(* CODESYS project PS_DcUpsEC_3.library
   Author: SAC
   Placeholder: PS_DcUpsEC
   Title: PS_DcUpsEC
   Version: 3.0
   Description: Function blocks for DC Uninterruptible Power Supplies with EtherCAT Interface
   Company: Phoenix Contact GmbH & Co.KG

Project tree, tasks and I/O mapping:
  libraries: Tc2_EtherCAT, * (Beckhoff Automation GmbH); Tc2_Standard, * (Beckhoff Automation GmbH); Tc2_System, * (Beckhoff Automation GmbH); Tc3_Module, * (Beckhoff Automation GmbH)
  DUTs/
    data type PS_CYCLIC_DATA
    data type PS_STATUS_FUNCTIONS
    data type PS_STATUS_INTERFACE
  GVLs/
  POUs/
    function block PS_Q4_DcUpsEC_Cyclic_3 [ST]: NewAlarmHandling, OldAlarmHandling
    function block PS_Q4_DcUpsEC_Param_1 [ST]
  Version/
    global variables Global_Version
  VISUs/
*)

// DUTs/PS_CYCLIC_DATA
TYPE PS_CYCLIC_DATA :
STRUCT
	srStatus_Functions  : PS_STATUS_FUNCTIONS;  (*Collection OF status signals*)        
	srStatus_Interface  : PS_STATUS_INTERFACE;  (*Collection OF interface signals*)        
	wInputVoltage       : WORD;         (*Input voltage in mV*)        
	wInputCurrent       : WORD;         (*Input current in mA*)        
	wOutputVoltage      : WORD;         (*Output voltage in mV*)        
	wOutputCurrent      : WORD;         (*Output current in mA*)        
	wBatteryVoltage     : WORD;         (*Battery voltage in mV*)        
	wBatteryChargeCurrent   : WORD;     (*Battery charge current in mA*)        
	wBatteryTemperature     : WORD;     (*Battery temperature in K*)        
	wDeviceTemperature      : WORD;     (*Device temperature in K*)        
	dwSocRemainingTime      : DWORD;    (*Remaining time in seconds*)        
	wSocRemainingTimePC_Shutdown: WORD; (*Remaining time until PC shutdown in s*)        
	wBatRemainingLifetime   : WORD;     (*Remaining lifetime in days*)
END_STRUCT
END_TYPE

// DUTs/PS_STATUS_FUNCTIONS
TYPE PS_STATUS_FUNCTIONS :
STRUCT
	xStartUpActive      : BOOL; (*Device is starting*)        
	xMainPowerModeActive: BOOL; (*Device is in mains mode*)        
	xBatteryModeActive  : BOOL; (*Device is in battery mode*)        
	xOutput             : BOOL; (*Output OF device is on/off*)        
	xBoost              : BOOL; (*Device is in boost mode*)        
	xChargerOn          : BOOL; (*Charger OF device is on/off*)        
	xBatteryComActive   : BOOL; (*Communcation to batteries is active/inactive*)        
	xStatusBatCom       : BOOL; (*Status communcation to batteries: 0=adressing, 1=normal communication*)        
	xAutonomicStart     : BOOL; (*Autonomic start input is open/closed*)        
	xRemoteConnected    : BOOL; (*Remote DI connected/disconnected*)        
	xRemoteEnabled      : BOOL; (*Remote is enabled/disabled*)        
	xPSinBoostMode      : BOOL; (*Power supply is in boost mode*)        
	xPhoenixAddCharger  : BOOL; (*Phoenix Contact additional charger is connected*)        
	xServiceModeActive  : BOOL; (*Device is in service mode*)        
	xBatDelay1Active    : BOOL; (*Battery mode delay time 1 is active*)        
	xBatDelay2Active    : BOOL; (*Battery mode delay time 2 is active*)        
	xBatDelay3Active    : BOOL; (*Battery mode delay time 3 is active**)        
	xExternalCharger    : BOOL; (*External charger active/inactive*)        
	xBufferReady        : BOOL; (*Connected energy storage is ready to buffer*)        
	xButtonUse          : BOOL; (*Service button enabled/disabled*)        
	xSelectorSwitchUse  : BOOL; (*Selector switch enabled/disabled*)        
	xSystemTest         : BOOL; (*System test active/inactive*)        
	xBatCapTest         : BOOL; (*Battery capacity test active/inactive*)        
	xBatteryPresent     : BOOL; (*Energy storage connected/disconnected*)        
	xSOC_Initialized    : BOOL; (*State OF charge initialized*)        
	xTriggerLogData     : BOOL; (*New log data available*)
END_STRUCT
END_TYPE

// DUTs/PS_STATUS_INTERFACE
TYPE PS_STATUS_INTERFACE :
STRUCT
	xDO1            : BOOL; (*DO1 is active/inactive*)        
	xDO2            : BOOL; (*DO2 is active/inactive*)        
	xDO3            : BOOL; (*DO3 is active/inactive*)        
	xDI1            : BOOL; (*DI1 is active/inactive*)        
	xDI2            : BOOL; (*DI2 is active/inactive*)        
	xDI3            : BOOL; (*DI3 is active/inactive*)        
	xModeSelector1  : BOOL; (*mode selector switch 1*)        
	xModeSelector2  : BOOL; (*mode selector switch 2*)        
	xModeSelector3  : BOOL; (*mode selector switch 3*)        
	xModeSelector4  : BOOL; (*mode selector switch 4*)        
	xSwitchPressed  : BOOL; (*Service button pressed/NOT pressed*)        
	xGreenLED       : BOOL; (*Green LED is on/off*)        
	xYellowLED      : BOOL; (*Yellow LED is on/off*)        
	xRedLED         : BOOL; (*Red LED is on/off*)        
	xBargraphRed    : BOOL; (*Red bargraph LED is on/off*)        
	xBargraphGreen1 : BOOL; (*Green bargraph LED 1 is on/off*)        
	xBargraphGreen2 : BOOL; (*Green bargraph LED 2 is on/off*)        
	xBargraphGreen3 : BOOL; (*Green bargraph LED 3 is on/off*)        
	xBargraphGreen4 : BOOL; (*Green bargraph LED 4 is on/off*)        
	xBargraphGreen5 : BOOL; (*Green bargraph LED 5 is on/off*)
	xSFB_Input		: BOOL;	(*SFB input is active/inactive*)
END_STRUCT
END_TYPE

// Version/Global_Version
{attribute 'TcGenerated'}
{attribute 'no-analysis'}
{attribute 'linkalways'}
// This function has been automatically generated from the project information.
VAR_GLOBAL CONSTANT
	{attribute 'const_non_replaced'}
	stLibVersion_PS_DcUpsEC : ST_LibVersion := (iMajor := 3, iMinor := 0, iBuild := 0, iRevision := 0, sVersion := '3.0');
END_VAR

// POUs/PS_Q4_DcUpsEC_Cyclic_3
{attribute 'hide_all_locals'}
FUNCTION_BLOCK PS_Q4_DcUpsEC_Cyclic_3
(*
wDiagCode	wAddDiagCode 	Description
16#0000		16#0000			Function block is inactive
16#8000		16#0000			Function block is active and without errors
*)
VAR_INPUT
	xActivate	: BOOL;		// TRUE: Activates function block
	arrInputPD	: ARRAY [0..30] OF WORD;	// Connect Multilink of TxPDO here
	tTimeout	: TIME := t#15s;	// Timeout value for communication timeout. Default t#15s.
END_VAR
VAR_OUTPUT
	xActive		: BOOL; // TRUE: Function block is working
	xError		: BOOL; // TRUE: An error occured at function block
	wDiagCode	: WORD; // Diagnosis Code of funtcion block error
	wAddDiagCode: WORD;	// Additional information about Diagnosis Code
	wOutputVoltage	: WORD; // Output Voltage of UPS in mV
	wOutputCurrent	: WORD; // Output Current of UPS in mA
	xBatModeActive	: BOOL; // TRUE: UPS is in Battery Mode
	udtDataStruct	: PS_CYCLIC_DATA; // Data structure contains voltages, currents, temperatures and remaining times
	xAlarm : BOOL; // TRUE: An alarm occured on the system
	xWarning : BOOL; // TRUE: An warning occured on the system
	xReplaceBattery : BOOL; // TRUE: Battery has to be replaced
	udtDiag : ARRAY[0..15] OF STRING; // Array of Alarm/Warning messages
END_VAR
VAR 
	(*_xyz - internal variables*)
	_wProcessAlarms : WORD;
	_dwUPSDiagnosis : DWORD;
	_dwBatAlarms : ARRAY[1..5] OF DWORD;
	_dwChargerAlarms : DWORD;
	_nI, _nK, _nM : INT;
	_xWarning: BOOL;
	_xAlarm: BOOL;
	_udtDiag : ARRAY[0..15] OF STRING;;
	_udtDeleteDiag : ARRAY[0..15] OF STRING; 
	_udtDelDataStruct	: PS_CYCLIC_DATA;
	_xBatModeActive: BOOL;
	_xReplaceBattery: BOOL;
	_fbTON : TON;
	_wBatteryVoltageOld	: WORD;
	_wInputVoltageOld : WORD;
	_wInputCurrentOld : WORD;
	_wOutputVoltageOld : WORD;
	_wOutputCurrentOld : WORD;
	_dwSocRemainingTimeOld :DWORD;	
	_xError : BOOL;
	_wDiagCode : WORD;
	_wAddDiagCode : WORD;
	_iNoOfActiveAlarms: INT;
	_iAlarmTypes: INT;
	_iAlarm_ID: INT;
	_iDevice_ID: INT;
	_arrAlarmBuffer : ARRAY [0..15] OF DWORD;
	_xNewAlarm : BOOL;
END_VAR

IF  xActivate THEN
	xActive := TRUE;
	_xError := FALSE;
	_wDiagCode := 16#8000;
	_wAddDiagCode := 16#0000;
	

	//-------------------------------------------------------------------------------
	
	// copy process alarms
	_wProcessAlarms := arrInputPD[16];
	// copy diagnosis alarms
	_dwUPSDiagnosis := SHL(WORD_TO_DWORD(arrInputPD[18]),DWORD#16);;
	_dwUPSDiagnosis := _dwUPSDiagnosis OR WORD_TO_DWORD(arrInputPD[17]);
	// Battery 1 Alarms
	_dwBatAlarms[1] := SHL(WORD_TO_DWORD(arrInputPD[20]),DWORD#16);;
	_dwBatAlarms[1] := _dwBatAlarms[1] OR WORD_TO_DWORD(arrInputPD[19]);
	// Battery 2 Alarms
	_dwBatAlarms[2] := SHL(WORD_TO_DWORD(arrInputPD[22]),DWORD#16);;
	_dwBatAlarms[2] := _dwBatAlarms[2] OR WORD_TO_DWORD(arrInputPD[21]);
	// Battery 3 Alarms
	_dwBatAlarms[3] := SHL(WORD_TO_DWORD(arrInputPD[24]),DWORD#16);;
	_dwBatAlarms[3] := _dwBatAlarms[3] OR WORD_TO_DWORD(arrInputPD[23]);
	// Battery 4 Alarms
	_dwBatAlarms[4] := SHL(WORD_TO_DWORD(arrInputPD[26]),DWORD#16);;
	_dwBatAlarms[4] := _dwBatAlarms[4] OR WORD_TO_DWORD(arrInputPD[25]);
	// Battery 5 Alarms
	_dwBatAlarms[5] := SHL(WORD_TO_DWORD(arrInputPD[28]),DWORD#16);;
	_dwBatAlarms[5] := _dwBatAlarms[5] OR WORD_TO_DWORD(arrInputPD[27]);
	// Charger Alarms
	_dwChargerAlarms := SHL(WORD_TO_DWORD(arrInputPD[30]),DWORD#16);;
	_dwChargerAlarms := _dwChargerAlarms OR WORD_TO_DWORD(arrInputPD[29]);
	

	//-------------------------------------------------------------------------------
	// build status functions
	udtDataStruct.srStatus_Functions.xStartUpActive 	:= arrInputPD[0].0;
	udtDataStruct.srStatus_Functions.xMainPowerModeActive := arrInputPD[0].1;
	udtDataStruct.srStatus_Functions.xBatteryModeActive := arrInputPD[0].2;
	udtDataStruct.srStatus_Functions.xOutput            := arrInputPD[0].3;        
	udtDataStruct.srStatus_Functions.xBoost             := arrInputPD[0].4;        
	udtDataStruct.srStatus_Functions.xChargerOn         := arrInputPD[0].5;        
	udtDataStruct.srStatus_Functions.xBatteryComActive  := arrInputPD[0].6;        
	udtDataStruct.srStatus_Functions.xStatusBatCom      := arrInputPD[0].7;        
	udtDataStruct.srStatus_Functions.xAutonomicStart    := arrInputPD[0].8;        
	udtDataStruct.srStatus_Functions.xRemoteConnected   := arrInputPD[0].9;        
	udtDataStruct.srStatus_Functions.xRemoteEnabled     := arrInputPD[0].10;        
	udtDataStruct.srStatus_Functions.xPSinBoostMode     := arrInputPD[0].11;  
    (*RESERVED := arrInputPD[0].12;*)  
	udtDataStruct.srStatus_Functions.xPhoenixAddCharger := arrInputPD[0].13;        
	udtDataStruct.srStatus_Functions.xServiceModeActive := arrInputPD[0].14;        
	udtDataStruct.srStatus_Functions.xBatDelay1Active   := arrInputPD[0].15;        
	udtDataStruct.srStatus_Functions.xBatDelay2Active   := arrInputPD[1].0;        
	udtDataStruct.srStatus_Functions.xBatDelay3Active   := arrInputPD[1].1;        
	udtDataStruct.srStatus_Functions.xExternalCharger   := arrInputPD[1].2;        
	udtDataStruct.srStatus_Functions.xBufferReady       := arrInputPD[1].3;        
	udtDataStruct.srStatus_Functions.xButtonUse         := arrInputPD[1].4;        
	udtDataStruct.srStatus_Functions.xSelectorSwitchUse := arrInputPD[1].5;        
	udtDataStruct.srStatus_Functions.xSystemTest        := arrInputPD[1].6;        
	udtDataStruct.srStatus_Functions.xBatCapTest        := arrInputPD[1].7;        
	udtDataStruct.srStatus_Functions.xBatteryPresent    := arrInputPD[1].8;        
	udtDataStruct.srStatus_Functions.xSOC_Initialized 	:= arrInputPD[1].9;        
	udtDataStruct.srStatus_Functions.xTriggerLogData 	:= arrInputPD[1].10;
	
	//Build status interface
	udtDataStruct.srStatus_Interface.xDO1					:= arrInputPD[2].0; (* STATUS_INTERFACE Bit 0 *)
	udtDataStruct.srStatus_Interface.xDO2					:= arrInputPD[2].1; (* STATUS_INTERFACE Bit 1 *)
	udtDataStruct.srStatus_Interface.xDO3					:= arrInputPD[2].2; (* STATUS_INTERFACE Bit 2 *)
	udtDataStruct.srStatus_Interface.xDI1					:= arrInputPD[2].4; (* STATUS_INTERFACE Bit 4 *)
	udtDataStruct.srStatus_Interface.xDI2					:= arrInputPD[2].5; (* STATUS_INTERFACE Bit 5 *)
	udtDataStruct.srStatus_Interface.xDI3					:= arrInputPD[2].6; (* STATUS_INTERFACE Bit 6 *)
	udtDataStruct.srStatus_Interface.xModeSelector1			:= arrInputPD[2].7; (* STATUS_INTERFACE Bit 7 *)
	udtDataStruct.srStatus_Interface.xModeSelector2			:= arrInputPD[2].8; (* STATUS_INTERFACE Bit 8 *)
	udtDataStruct.srStatus_Interface.xModeSelector3			:= arrInputPD[2].9; (* STATUS_INTERFACE Bit 9 *)
	udtDataStruct.srStatus_Interface.xModeSelector4			:= arrInputPD[2].10; (* STATUS_INTERFACE Bit 10 *)
	udtDataStruct.srStatus_Interface.xSwitchPressed			:= arrInputPD[2].11; (* STATUS_INTERFACE Bit 11 *)
	udtDataStruct.srStatus_Interface.xGreenLED				:= arrInputPD[2].12; (* STATUS_INTERFACE Bit 12 *)
	udtDataStruct.srStatus_Interface.xYellowLED				:= arrInputPD[2].13; (* STATUS_INTERFACE Bit 13 *)
	udtDataStruct.srStatus_Interface.xRedLED				:= arrInputPD[2].14; (* STATUS_INTERFACE Bit 14 *)
	udtDataStruct.srStatus_Interface.xBargraphRed			:= arrInputPD[2].15; (* STATUS_INTERFACE Bit 15 *)
	udtDataStruct.srStatus_Interface.xBargraphGreen1		:= arrInputPD[3].0; (* STATUS_INTERFACE Bit 16 *)
	udtDataStruct.srStatus_Interface.xBargraphGreen2		:= arrInputPD[3].1; (* STATUS_INTERFACE Bit 17 *)
	udtDataStruct.srStatus_Interface.xBargraphGreen3		:= arrInputPD[3].2; (* STATUS_INTERFACE Bit 18 *)
	udtDataStruct.srStatus_Interface.xBargraphGreen4		:= arrInputPD[3].3; (* STATUS_INTERFACE Bit 19 *)
	udtDataStruct.srStatus_Interface.xBargraphGreen5		:= arrInputPD[3].4; (* STATUS_INTERFACE Bit 20 *)
	udtDataStruct.srStatus_Interface.xSFB_Input				:= arrInputPD[3].5; (* STATUS_INTERFACE Bit 21 *)
	
	//copy values into data structure
	udtDataStruct.wInputVoltage := arrInputPD[4];
	udtDataStruct.wInputCurrent := arrInputPD[5];
	udtDataStruct.wOutputVoltage := arrInputPD[6];
	wOutputVoltage := arrInputPD[6];
	udtDataStruct.wOutputCurrent := arrInputPD[7];
	wOutputCurrent := arrInputPD[7];
	udtDataStruct.wBatteryVoltage := arrInputPD[8];
	udtDataStruct.wBatteryChargeCurrent := arrInputPD[9];
	udtDataStruct.wBatteryTemperature := arrInputPD[10];
	udtDataStruct.wDeviceTemperature := arrInputPD[11];
	
	udtDataStruct.dwSocRemainingTime := SHL(WORD_TO_DWORD(arrInputPD[13]),DWORD#16);
	udtDataStruct.dwSocRemainingTime := udtDataStruct.dwSocRemainingTime OR WORD_TO_DWORD(arrInputPD[12]);
	
	udtDataStruct.wSocRemainingTimePC_Shutdown := arrInputPD[14];
	udtDataStruct.wBatRemainingLifetime := arrInputPD[15];
	
	//-------------------------------------------------------------------------------
	// evaluate alarms and warnings
	// initialize
	_nI := 0; // reset alarm counter
	_xWarning := FALSE;
	_xAlarm := FALSE;
	_udtDiag := _udtDeleteDiag;
	_xBatModeActive := FALSE;
	_xReplaceBattery := FALSE;

	

	// evaluate process alarms
	IF _wProcessAlarms.0 THEN
		_udtDiag[_nI] := 'Warning: Any user counter exceeded';
		_nI := _nI + 1;
		_xWarning := TRUE;
	END_IF
	IF _wProcessAlarms.1 THEN
		_udtDiag[_nI] := 'Warning: User threshold battery voltage exceeded';
		_nI := _nI + 1;
		_xWarning := TRUE;
	END_IF
	IF _wProcessAlarms.2 THEN
		_udtDiag[_nI] := 'Warning: User threshold SOC [%] low exceeded';
		_nI := _nI + 1;
		_xWarning := TRUE;
	END_IF
	IF _wProcessAlarms.3 THEN
		_udtDiag[_nI] := 'Warning: User threshold SOC [min] low exceeded';
		_nI := _nI + 1;
		_xWarning := TRUE;
	END_IF
	IF _wProcessAlarms.4 THEN
		_udtDiag[_nI] := 'Battery mode active';
		_nI := _nI + 1;
		_xWarning := TRUE;
		_xBatModeActive := TRUE;
	END_IF
	IF _wProcessAlarms.5 THEN
		_udtDiag[_nI] := 'Capacity test active';
		_nI := _nI + 1;
		_xWarning := TRUE;
	END_IF
	IF _wProcessAlarms.6 THEN
		_udtDiag[_nI] := 'Shutdown event triggered';
		_nI := _nI + 1;
		_xWarning := TRUE;
	END_IF
	IF _wProcessAlarms.7 THEN
		_udtDiag[_nI] := 'Service mode active';
		_nI := _nI + 1;
		_xWarning := TRUE;
	END_IF
	
	// UPS diagnosis alarms
	IF _dwUPSDiagnosis.2 THEN
		_udtDiag[_nI] := 'Alarm: Overload cutoff';
		_nI := _nI + 1;
		_xAlarm := TRUE;
	END_IF
	IF _dwUPSDiagnosis.5 THEN
		_udtDiag[_nI] := 'Alarm: Internal fault';
		_nI := _nI + 1;
		_xAlarm := TRUE;
	END_IF
	IF _dwUPSDiagnosis.6 THEN
		_udtDiag[_nI] := 'Alarm: Battery technologies different';
		_nI := _nI + 1;
		_xAlarm := TRUE;
	END_IF
	IF _dwUPSDiagnosis.7 THEN
		_udtDiag[_nI] := 'Alarm: Battery capacities different';
		_nI := _nI + 1;
		_xAlarm := TRUE;
	END_IF
	IF _dwUPSDiagnosis.8 THEN
		_udtDiag[_nI] := 'Alarm: Battery capacity test negative';
		_nI := _nI + 1;
		_xAlarm := TRUE;
	END_IF
	IF _dwUPSDiagnosis.9 THEN
		_udtDiag[_nI] := 'Alarm: Battery capacity too high';
		_nI := _nI + 1;
		_xAlarm := TRUE;
	END_IF
	IF _dwUPSDiagnosis.10 THEN
		_udtDiag[_nI] := 'Alarm: Battery capacity too low';
		_nI := _nI + 1;
		_xAlarm := TRUE;
	END_IF
	IF _dwUPSDiagnosis.11 THEN
		_udtDiag[_nI] := 'Alarm: Temperature drop between batteries too high';
		_nI := _nI + 1;
		_xAlarm := TRUE;
	END_IF
	IF _dwUPSDiagnosis.12 THEN
		_udtDiag[_nI] := 'Alarm: Battery quality check negative';
		_nI := _nI + 1;
		_xAlarm := TRUE;
	END_IF
	IF _dwUPSDiagnosis.13 THEN
		_udtDiag[_nI] := 'Alarm: End of Lifetime reached';
		_nI := _nI + 1;
		_xAlarm := TRUE;
	END_IF
	IF _dwUPSDiagnosis.14 THEN
		_udtDiag[_nI] := 'Alarm: No battery detected';
		_nI := _nI + 1;
		_xAlarm := TRUE;
	END_IF
	IF _dwUPSDiagnosis.16 THEN
		_udtDiag[_nI] := 'Alarm: Replace Battery';
		_nI := _nI + 1;
		_xAlarm := TRUE;
		_xReplaceBattery := TRUE;
	END_IF
	
			
	(*If VC05 Device detected then start new data evaluation*)
	IF _dwBatAlarms[1].31 THEN
		NewAlarmHandling();
	(*If device <VC05 detected then start old data evaluation*)
	ELSE	
		OldAlarmHandling();
	END_IF;
		
	// If functionm block doesn't receive any new process data throw error and timeout diag code
	_fbTON(IN:= (udtDataStruct.wBatteryVoltage = _wBatteryVoltageOld AND
				udtDataStruct.wInputVoltage = _wInputVoltageOld AND
				udtDataStruct.wInputCurrent = _wInputCurrentOld AND
				udtDataStruct.wOutputVoltage = _wOutputVoltageOld AND
				udtDataStruct.wOutputCurrent = 	_wOutputCurrentOld AND
				udtDataStruct.dwSocRemainingTime = _dwSocRemainingTimeOld), 
				PT:=tTimeout);
	IF _fbTON.Q THEN
		_xError := TRUE;
		_wDiagCode := 16#C415;
		_wAddDiagCode := 16#0000;
	END_IF
	
	_wBatteryVoltageOld := udtDataStruct.wBatteryVoltage;
	_wInputVoltageOld := udtDataStruct.wInputVoltage;
	_wInputCurrentOld := udtDataStruct.wInputCurrent;
	_wOutputVoltageOld := udtDataStruct.wOutputVoltage;
	_wOutputCurrentOld := udtDataStruct.wOutputCurrent;
	_dwSocRemainingTimeOld := udtDataStruct.dwSocRemainingTime;
	
	// write outputs
	xError := _xError;
	wDiagCode := _wDiagCode;
	wAddDiagCode := _wAddDiagCode;
	xAlarm := _xAlarm;
	xWarning := _xWarning;
	udtDiag := _udtDiag;
	xBatModeActive := _xBatModeActive;
	xReplaceBattery := _xReplaceBattery;
	
	
ELSE
	//reset all outputs
	xActive := FALSE;
	wDiagCode := 16#0000;
	wAddDiagCode := 16#0000;
	xAlarm := FALSE;
	xWarning := FALSE;
	xBatModeActive := FALSE;
	xReplaceBattery := FALSE;
	wOutputVoltage := WORD#0;
	wOutputCurrent := WORD#0;
	udtDataStruct := _udtDelDataStruct;
	udtDiag := _udtDeleteDiag;
	
END_IF

METHOD INTERNAL NewAlarmHandling : BOOL
VAR_INPUT
END_VAR
VAR
	strBattery1 : STRING := 'Battery 1: ';
	strBattery2 : STRING := 'Battery 2: ';
	strBattery3 : STRING := 'Battery 3: ';
	strBattery4 : STRING := 'Battery 4: ';
	strBattery5 : STRING := 'Battery 5: ';
	strCharger  : STRING := 'QUINT4 Charger: ';
	strPowSup   : STRING := 'QUINT4 Power Supply: ';
	
	strEvent : STRING := 'Warning: ';
	strMR	 : STRING := 'Maintenance required: ';
	strMD	 : STRING := 'Maintenance demanded: ';
	strDiag  : STRING := 'Alarm: ';
	
	
END_VAR
// Evaluate data, how many alarms occured
_iNoOfActiveAlarms.0 := _dwBatAlarms[1].0;
_iNoOfActiveAlarms.1 := _dwBatAlarms[1].1;
_iNoOfActiveAlarms.2 := _dwBatAlarms[1].2;
_iNoOfActiveAlarms.3 := _dwBatAlarms[1].3;
_iNoOfActiveAlarms.4 := _dwBatAlarms[1].4;
		
IF _iNoOfActiveAlarms <> 0 THEN

//--Check if new alarms are available, if yes, save them----------------------	
	FOR _nK := 1 TO _iNoOfActiveAlarms DO
		_xNewAlarm := TRUE;
		IF _arrAlarmBuffer[_nK-1] = _dwBatAlarms[1] THEN
			_xNewAlarm := FALSE;	(*Received Alarm is already saved*)
			EXIT;
		END_IF
		
	END_FOR
	
	IF _xNewAlarm THEN
		_arrAlarmBuffer[_nM] :=  _dwBatAlarms[1];
		_nM := _nM + 1;
		IF _nM > _iNoOfActiveAlarms-1 THEN
			_nM := 0;
		END_IF
	END_IF
//---------------------------------------------------------------------------	
//--Alarm evaluation---------------------------------------------------------	
	FOR _nK := 0 TO _iNoOfActiveAlarms-1 DO
		// DeviceID: 1 - 5: Battery 6: QUITN4-Charger 7: QUINT4 - PS
		_iDevice_ID.0 := _arrAlarmBuffer[_nK].15;
		_iDevice_ID.1 := _arrAlarmBuffer[_nK].16;
		_iDevice_ID.2 := _arrAlarmBuffer[_nK].17;
		_iDevice_ID.3 := _arrAlarmBuffer[_nK].18;
		_iDevice_ID.4 := _arrAlarmBuffer[_nK].19;
		_iDevice_ID.5 := _arrAlarmBuffer[_nK].20;
		_iDevice_ID.6 := _arrAlarmBuffer[_nK].21;
		_iDevice_ID.7 := _arrAlarmBuffer[_nK].22;
		_iDevice_ID.8 := _arrAlarmBuffer[_nK].23;
		_iDevice_ID.9 := _arrAlarmBuffer[_nK].24;
		_iDevice_ID.10 := _arrAlarmBuffer[_nK].25;
		_iDevice_ID.11 := _arrAlarmBuffer[_nK].26;
		_iDevice_ID.12 := _arrAlarmBuffer[_nK].27;
		_iDevice_ID.13 := _arrAlarmBuffer[_nK].28;
		_iDevice_ID.14 := _arrAlarmBuffer[_nK].29;
		_iDevice_ID.15 := _arrAlarmBuffer[_nK].30;

		// 1 : Process Alarm / Event, 2: Maintenance required, 3: Maintenance demand, 4: Diagnosis Alarm
		_iAlarmTypes.0 := _arrAlarmBuffer[_nK].5;
		_iAlarmTypes.1 := _arrAlarmBuffer[_nK].6;
		_iAlarmTypes.2 := _arrAlarmBuffer[_nK].7;
		
		// Alarm ID according to the spec
		_iAlarm_ID.0 := _arrAlarmBuffer[_nK].8;
		_iAlarm_ID.1 := _arrAlarmBuffer[_nK].9;
		_iAlarm_ID.2 := _arrAlarmBuffer[_nK].10;
		_iAlarm_ID.3 := _arrAlarmBuffer[_nK].11;
		_iAlarm_ID.4 := _arrAlarmBuffer[_nK].12;
		_iAlarm_ID.5 := _arrAlarmBuffer[_nK].13;
		_iAlarm_ID.6 := _arrAlarmBuffer[_nK].14;
		

		// Which Alarm type
		CASE _iAlarmTypes OF
			1 : // Process Alarm / Event
				_udtDiag[_nI] := strEvent;
				_xWarning := TRUE;
				
				//Which device
				CASE _iDevice_ID OF
					1..5: // Battery 1-5, currently no warnings available
							;
			
					6: // QUINT4 Charger, currently no warnings available
							;
					
					7: // QUINT4 Power Supply
						_udtDiag[_nI] := CONCAT(strEvent,strPowSup);
						
						CASE _iAlarm_ID OF
							1: // Output voltage warning
								_udtDiag[_nI] := CONCAT(_udtDiag[_nI],'Output voltage warning');
							
							8: // PS configuration error
								_udtDiag[_nI] := CONCAT(_udtDiag[_nI],'PS configuration error');

							9: // Output power warning
								_udtDiag[_nI] := CONCAT(_udtDiag[_nI],'Output power warning');
							
							10: // Prewarning temperature derating
								_udtDiag[_nI] := CONCAT(_udtDiag[_nI],'Prewarning temperature derating');
							
							11: // Two phase operation
								_udtDiag[_nI] := CONCAT(_udtDiag[_nI],'Two phase operation');
							
							12:	// Predictive maintenance recommended (Remaining Lifetime)
								_udtDiag[_nI] := CONCAT(_udtDiag[_nI],'Predictive maintenance recommended (Remaining Lifetime)');

						END_CASE
				END_CASE
				_nI := _nI + 1;		// increase Diag array index		

			2: // Maintenance required
				_udtDiag[_nI] := strMR;
				//NOT IN USE
				

			3: // Maintenance demand
				_udtDiag[_nI] := strMD;
				// NOT IN USE
				

			4: // Diagnosis Alarm 
				_udtDiag[_nI] := strDiag;
				_xAlarm := TRUE;
				
				//Which device
				CASE _iDevice_ID OF
					1: // Battery 1
						_udtDiag[_nI] := CONCAT(strDiag,strBattery1);
						
						CASE _iAlarm_ID OF
							0: // Undervoltage
								_udtDiag[_nI] := CONCAT(_udtDiag[_nI],'Undervoltage');
								
							1: // overvoltage
								_udtDiag[_nI] := CONCAT(_udtDiag[_nI],'Overvoltage');

							3: // overTempLow
								_udtDiag[_nI] := CONCAT(_udtDiag[_nI],'Overtemperature (+40 degrees)');

							4: // overTempHigh
								_udtDiag[_nI] := CONCAT(_udtDiag[_nI],'Overtemperature (+60 degrees)');

							5: // internalFault
								_udtDiag[_nI] := CONCAT(_udtDiag[_nI],'Internal Fault');

							14: // no or UnknownDev
								_udtDiag[_nI] := CONCAT(_udtDiag[_nI],'No or unknown Device detected');

							15: // underTemp
								_udtDiag[_nI] := CONCAT(_udtDiag[_nI],'Undertemperature');

							17: // fuseBlown
								_udtDiag[_nI] := CONCAT(_udtDiag[_nI],'Fuse blown');

							18: // comFault
								_udtDiag[_nI] := CONCAT(_udtDiag[_nI],'Communication fault');
							
						END_CASE
			
					2: // Battery 2
						_udtDiag[_nI] := CONCAT(strDiag,strBattery2);
						
						CASE _iAlarm_ID OF
							0: // Undervoltage
								_udtDiag[_nI] := CONCAT(_udtDiag[_nI],'Undervoltage');
								
							1: // overvoltage
								_udtDiag[_nI] := CONCAT(_udtDiag[_nI],'Overvoltage');

							3: // overTempLow
								_udtDiag[_nI] := CONCAT(_udtDiag[_nI],'Overtemperature (+40 degrees)');

							4: // overTempHigh
								_udtDiag[_nI] := CONCAT(_udtDiag[_nI],'Overtemperature (+60 degrees)');

							5: // internalFault
								_udtDiag[_nI] := CONCAT(_udtDiag[_nI],'Internal Fault');

							14: // no or UnknownDev
								_udtDiag[_nI] := CONCAT(_udtDiag[_nI],'No or unknown Device detected');

							15: // underTemp
								_udtDiag[_nI] := CONCAT(_udtDiag[_nI],'Undertemperature');

							17: // fuseBlown
								_udtDiag[_nI] := CONCAT(_udtDiag[_nI],'Fuse blown');

							18: // comFault
								_udtDiag[_nI] := CONCAT(_udtDiag[_nI],'Communication fault');
							
						END_CASE						
			
					3: // Battery 3
						_udtDiag[_nI] := CONCAT(strDiag,strBattery3);
						
						CASE _iAlarm_ID OF
							0: // Undervoltage
								_udtDiag[_nI] := CONCAT(_udtDiag[_nI],'Undervoltage');
								
							1: // overvoltage
								_udtDiag[_nI] := CONCAT(_udtDiag[_nI],'Overvoltage');

							3: // overTempLow
								_udtDiag[_nI] := CONCAT(_udtDiag[_nI],'Overtemperature (+40 degrees)');

							4: // overTempHigh
								_udtDiag[_nI] := CONCAT(_udtDiag[_nI],'Overtemperature (+60 degrees)');

							5: // internalFault
								_udtDiag[_nI] := CONCAT(_udtDiag[_nI],'Internal Fault');

							14: // no or UnknownDev
								_udtDiag[_nI] := CONCAT(_udtDiag[_nI],'No or unknown Device detected');

							15: // underTemp
								_udtDiag[_nI] := CONCAT(_udtDiag[_nI],'Undertemperature');

							17: // fuseBlown
								_udtDiag[_nI] := CONCAT(_udtDiag[_nI],'Fuse blown');

							18: // comFault
								_udtDiag[_nI] := CONCAT(_udtDiag[_nI],'Communication fault');
							
						END_CASE						
					
					4: // Battery 4
						_udtDiag[_nI] := CONCAT(strDiag,strBattery4);
						
						CASE _iAlarm_ID OF
							0: // Undervoltage
								_udtDiag[_nI] := CONCAT(_udtDiag[_nI],'Undervoltage');
								
							1: // overvoltage
								_udtDiag[_nI] := CONCAT(_udtDiag[_nI],'Overvoltage');

							3: // overTempLow
								_udtDiag[_nI] := CONCAT(_udtDiag[_nI],'Overtemperature (+40 degrees)');

							4: // overTempHigh
								_udtDiag[_nI] := CONCAT(_udtDiag[_nI],'Overtemperature (+60 degrees)');

							5: // internalFault
								_udtDiag[_nI] := CONCAT(_udtDiag[_nI],'Internal Fault');

							14: // no or UnknownDev
								_udtDiag[_nI] := CONCAT(_udtDiag[_nI],'No or unknown Device detected');

							15: // underTemp
								_udtDiag[_nI] := CONCAT(_udtDiag[_nI],'Undertemperature');

							17: // fuseBlown
								_udtDiag[_nI] := CONCAT(_udtDiag[_nI],'Fuse blown');

							18: // comFault
								_udtDiag[_nI] := CONCAT(_udtDiag[_nI],'Communication fault');
							
						END_CASE						
					
					5: // Battery 5
						_udtDiag[_nI] := CONCAT(strDiag,strBattery4);
						
						CASE _iAlarm_ID OF
							0: // Undervoltage
								_udtDiag[_nI] := CONCAT(_udtDiag[_nI],'Undervoltage');
								
							1: // overvoltage
								_udtDiag[_nI] := CONCAT(_udtDiag[_nI],'Overvoltage');

							3: // overTempLow
								_udtDiag[_nI] := CONCAT(_udtDiag[_nI],'Overtemperature (+40 degrees)');

							4: // overTempHigh
								_udtDiag[_nI] := CONCAT(_udtDiag[_nI],'Overtemperature (+60 degrees)');

							5: // internalFault
								_udtDiag[_nI] := CONCAT(_udtDiag[_nI],'Internal Fault');

							14: // no or UnknownDev
								_udtDiag[_nI] := CONCAT(_udtDiag[_nI],'No or unknown Device detected');

							15: // underTemp
								_udtDiag[_nI] := CONCAT(_udtDiag[_nI],'Undertemperature');

							17: // fuseBlown
								_udtDiag[_nI] := CONCAT(_udtDiag[_nI],'Fuse blown');

							18: // comFault
								_udtDiag[_nI] := CONCAT(_udtDiag[_nI],'Communication fault');
							
						END_CASE						
					
					6: // QUINT4 Charger
						_udtDiag[_nI] := CONCAT(strDiag,strCharger);
						
						CASE _iAlarm_ID OF
						0: // Undervoltage 
							_udtDiag[_nI] := CONCAT(_udtDiag[_nI],'No AC input voltage');
							
						14: // no or UnknownDev
							_udtDiag[_nI] := CONCAT(_udtDiag[_nI],'No or unknown Device detected');

						18: // comFault
							_udtDiag[_nI] := CONCAT(_udtDiag[_nI],'Communication fault');						

						END_CASE						
					
					7: // QUINT4 Power Supply
						_udtDiag[_nI] := CONCAT(strDiag,strPowSup);
						
						CASE _iAlarm_ID OF
						0: // Undervoltage 
							_udtDiag[_nI] := CONCAT(_udtDiag[_nI],'No AC input voltage');
						
							
						1: // Overvoltage
							_udtDiag[_nI] := CONCAT(_udtDiag[_nI],'Voltage limitation active (OVP)');
							
						2: // Overload	
							_udtDiag[_nI] := CONCAT(_udtDiag[_nI],'Overload');	
							
						14: // Unknown device detected 
							_udtDiag[_nI] := CONCAT(_udtDiag[_nI],'Unknown device detected');
						
						
						17: // FUSE MODE tripped
							_udtDiag[_nI] := CONCAT(_udtDiag[_nI],'FUSE MODE tripped');
						
						
						18: //	Communication fault 
							_udtDiag[_nI] := CONCAT(_udtDiag[_nI],'Communication fault');
						
							
						END_CASE
						
				END_CASE				
				_nI := _nI + 1;		// increase Diag array index
		END_CASE
	END_FOR
	
	
// If No of alarms = 0 then delete Alarm buffer	
ELSE
	FOR _nK := 0 TO 15 DO
		_arrAlarmBuffer[_nK] := 0;
	END_FOR	
END_IF
END_METHOD

METHOD INTERNAL OldAlarmHandling : BOOL
VAR_INPUT
END_VAR
// Battery alarms
FOR _nK := 1 TO 5 DO
	IF _dwBatAlarms[_nK].0 THEN
		_udtDiag[_nI] := CONCAT('Battery ', INT_TO_STRING(_nK));
		_udtDiag[_nI] := CONCAT(_udtDiag[_nI],': Voltage too low');
		_nI := _nI + 1;
		_xAlarm := TRUE;
	END_IF
	IF _dwBatAlarms[_nK].1 THEN
		_udtDiag[_nI] := CONCAT('Battery ', INT_TO_STRING(_nK));
		_udtDiag[_nI] := CONCAT(_udtDiag[_nI],': Voltage too high');
		_nI := _nI + 1;
		_xAlarm := TRUE;
	END_IF
	IF _dwBatAlarms[_nK].3 THEN
		_udtDiag[_nI] := CONCAT('Battery ', INT_TO_STRING(_nK));
		_udtDiag[_nI] := CONCAT(_udtDiag[_nI],': Warning: Temperature too high');
		_nI := _nI + 1;
		_xAlarm := TRUE;
	END_IF
	IF _dwBatAlarms[_nK].4 THEN
		_udtDiag[_nI] := CONCAT('Battery ', INT_TO_STRING(_nK));
		_udtDiag[_nI] := CONCAT(_udtDiag[_nI],': Temperature too high');
		_nI := _nI + 1;
		_xAlarm := TRUE;
	END_IF
	IF _dwBatAlarms[_nK].5 THEN
		_udtDiag[_nI] := CONCAT('Battery ', INT_TO_STRING(_nK));
		_udtDiag[_nI] := CONCAT(_udtDiag[_nI],': Internal fault');
		_nI := _nI + 1;
		_xAlarm := TRUE;
	END_IF
	IF _dwBatAlarms[_nK].14 THEN
		_udtDiag[_nI] := CONCAT('Battery ', INT_TO_STRING(_nK));
		_udtDiag[_nI] := CONCAT(_udtDiag[_nI],': No or unknown device detected');
		_nI := _nI + 1;
		_xAlarm := TRUE;
	END_IF
	IF _dwBatAlarms[_nK].15 THEN
		_udtDiag[_nI] := CONCAT('Battery ', INT_TO_STRING(_nK));
		_udtDiag[_nI] := CONCAT(_udtDiag[_nI],': Temperature too low');
		_nI := _nI + 1;
		_xAlarm := TRUE;
	END_IF
	IF _dwBatAlarms[_nK].17 THEN
		_udtDiag[_nI] := CONCAT('Battery ', INT_TO_STRING(_nK));
		_udtDiag[_nI] := CONCAT(_udtDiag[_nI],': Fuse blown');
		_nI := _nI + 1;
		_xAlarm := TRUE;
	END_IF
	IF _dwBatAlarms[_nK].18 THEN
		_udtDiag[_nI] := CONCAT('Battery ', INT_TO_STRING(_nK));
		_udtDiag[_nI] := CONCAT(_udtDiag[_nI],': Communication fault');
		_nI := _nI + 1;
		_xAlarm := TRUE;
	END_IF
END_FOR

// Charger Alarme
IF _dwChargerAlarms.0 THEN
	_udtDiag[_nI] := 'QUINT Charger Alarm: AC Input down';
	_nI := _nI + 1;
	_xAlarm := TRUE;
END_IF

IF _dwChargerAlarms.14 THEN
	_udtDiag[_nI] := 'QUINT Charger Alarm: Unknown device detected';
	_nI := _nI + 1;
	_xAlarm := TRUE;
END_IF

	IF _dwChargerAlarms.18 THEN
	_udtDiag[_nI] := 'QUINT Charger Alarm: Communication fault';
	_nI := _nI + 1;
	_xAlarm := TRUE;
END_IF;
END_METHOD

END_FUNCTION_BLOCK

// POUs/PS_Q4_DcUpsEC_Param_1
{attribute 'hide_all_locals'}
FUNCTION_BLOCK PS_Q4_DcUpsEC_Param_1
VAR_INPUT
	xActivate		: BOOL;		// TRUE: Activates function block
	sNetId			: STRING; 	// NetID of the Master
	uintSlaveAddr	: UINT;		// Slave address
	wIndex  		: WORD;		// Index to read from/write to 
	xReceive		: BOOL;
	udintReceiveLength	: UDINT;
	tTimeOutReading : TIME := T#500MS;
	xSend			: BOOL;
	udintSendLength	: UDINT;
	arrWriteParameter 	: ARRAY [0..7] OF DWORD; 
	tTimeOutWriting : TIME := T#500MS;
END_VAR

VAR_OUTPUT
	xActive			: BOOL; 	// TRUE: Function block is active
	xError			: BOOL;		// TRUE: Error while executing function block
	wDiagCode		: WORD;		// Diagnosis code of function block 
	wAddDiagCode	: WORD;		// Additional information to Diagnosis Code
	arrReadParameter 	: ARRAY [0..7] OF DWORD;

END_VAR
	
VAR_IN_OUT
	xBusy			: BOOL;		// TRUE: Baustein ist mit einer Operation beschäftigt
END_VAR

VAR
// for internal use only	
	// reading / writing execution
	_ReadParam: FB_EcCoESdoRead;		// FB to read data
	_WriteParam: FB_EcCoESdoWrite;		// FB to write data
	_sNetId: T_AmsNetId;				// NetID of connected Master
	_uintSlaveAddr: UINT;				// Slave address of connected slace
	_wIndex: WORD;						// Index of parameter for reading/writing
	_xReadCommand: BOOL;				// reading flag to execute reading function block
	_udintReadLength: UDINT;			// Length of variable to read	
	_xWriteCommand: BOOL;				// writing flag to execute writing function block
	_udintSendLength: UDINT;			// Length of variable to write 
	_xBusy : BOOL;						// function block is operatiing

	// management of execution
	_RTRIG_Read : R_TRIG;				// function block to detect rising edge of reading
	_RTRIG_Write : R_TRIG;				// function block to detect rising edge of writing	
	_xRead: BOOL;						// Reading flag detected, save for execution
	_xWrite: BOOL;						// Writing flag detected, save for execution
	_nI, _nK: INT;							// case loop variable	
	_arrReadBuffer : ARRAY [0..7] OF DWORD;
	_arrWriteBuffer : ARRAY [0..7] OF DWORD; 

	// copy to outputs
	_xActive: BOOL;						// function block is active
	_xError: BOOL;						// TRUE: an error occured
	_wDiagCode: WORD;					// diagnosis code in case of function block error
	_wAddDiagCode: WORD;				// additional information for diagnosis code


END_VAR


IF xActivate THEN
	_xActive := TRUE;


	// detect rising edges for reading / writing
	_RTRIG_Read(CLK:=xReceive);
	_RTRIG_Write(CLK:=xSend);
	
	//evaluate rising edges and save flag
	IF _RTRIG_Read.Q THEN
		_xRead := TRUE;		// Reset flag in case loop
		_xError := FALSE;
	END_IF
	IF _RTRIG_Write.Q THEN
		_xWrite := TRUE;	// Reset flag in case loop
		_xError := FALSE;
	END_IF
	
	
	CASE _nI OF
		0: 	// Init
			_wDiagCode := WORD#16#8000;
			_wAddDiagCode := WORD#16#0000;	
			_nI := 1;
		
		1:	// which command was set?
			IF _xRead THEN
				_xRead := FALSE;
				IF sNetID = '' OR uintSlaveAddr = 0 THEN
					_nK := _nI;
					_nI := 99;
				ELSE	
					_xBusy := TRUE;
					_nI := 10;
					_wDiagCode := WORD#16#8000;
					_wAddDiagCode := WORD#16#0000;		
					MEMSET(ADR(_arrReadBuffer),0,SIZEOF(_arrReadBuffer));			
				END_IF;	
			ELSIF _xWrite THEN
				_xWrite := FALSE;
				IF sNetID = '' OR uintSlaveAddr = 0 THEN
					_nK := _nI;
					_nI := 99;
				ELSE					
					_xBusy := TRUE;
					_nI := 20;
					_wDiagCode := WORD#16#8000;
					_wAddDiagCode := WORD#16#0000;	
				END_IF
			ELSE 
				_nI := _nI;		
			END_IF
			
		
		10: // reading execution
			_sNetId := sNetId;	
			_uintSlaveAddr := uintSlaveAddr;
			_wIndex := wIndex;
			_udintReadLength := udintReceiveLength;
			_xReadCommand := TRUE;
			_nI := 11;
			
		11: // check if function block is running
			IF _ReadParam.bBusy THEN
				_nI := 12;
			ELSIF _ReadParam.bError THEN
				_nK := _nI;
				_nI := 99;	
			ELSE
				_nI := _nI;	
			END_IF
	
		12: // wait until function block finished execution
			IF NOT _ReadParam.bBusy AND NOT _ReadParam.bError THEN
				arrReadParameter := _arrReadBuffer;	// copy read result to output variables
				_xReadCommand := FALSE;
				_xBusy := FALSE;
				_nI := 1;
			ELSIF _ReadParam.bError THEN
				_nK := _nI;
				_nI := 99;
			ELSE
				_nI := _nI;		
			END_IF	
		
		
		20: // writing execution
			_sNetId := sNetId;	
			_uintSlaveAddr := uintSlaveAddr;
			_wIndex := wIndex;
			_xWriteCommand := TRUE;
			_arrWriteBuffer := arrWriteParameter;
			_udintSendLength := udintSendLength;
			_nI := 21;
	
		21: // check if function block is running
			IF _WriteParam.bBusy THEN
				_nI := 22;
			ELSIF _WriteParam.bError THEN
				_nK := _nI;
				_nI := 99;	
			ELSE
				_nI := _nI;	
			END_IF
	
		22: // wait until function block finished execution
			IF NOT _WriteParam.bBusy AND NOT _WriteParam.bError THEN
				_arrWriteBuffer := arrWriteParameter;
				_xWriteCommand := FALSE;
				_xBusy := FALSE;
				_nI := 1;
			ELSIF _WriteParam.bError THEN
				_nK := _nI;
				_nI := 99;
			ELSE
				_nI := _nI;		
			END_IF	
			
			
		99: // Error case	
			CASE _nK OF
			1:	// Input error 	
				IF sNetID = ''  THEN
					_wDiagCode := 16#C110;
					_wAddDiagCode := 16#0002;
				ELSIF uintSlaveAddr = 0 THEN
					_wDiagCode := 16#C110;
					_wAddDiagCode := 16#0003;	
				ELSE
					_wDiagCode := 16#FFFF;		// unkown error
					_wAddDiagCode := 16#FFFF;	// unknown error
				END_IF;	
				_xError := TRUE;
				_nI := 1;
				
			11,12: // Read error
				_wDiagCode := 16#C350;
				_wAddDiagCode := UDINT_TO_WORD(_ReadParam.nErrId);
				_xReadCommand := FALSE;
				_xError := TRUE;
				_xBusy := FALSE;
				_nI := 1;
				
			21,22: // Write error
				_wDiagCode := 16#C351;
				_wAddDiagCode := UDINT_TO_WORD(_WriteParam.nErrId);
				_xWriteCommand := FALSE;
				_xError := TRUE;
				_xBusy := FALSE;
				_nI := 1;			
				
			ELSE
				_nI := 0;
				_nK := 0;	
			END_CASE
	END_CASE

ELSE
	_xActive := FALSE;
	_xError := FALSE;
	_wDiagCode := WORD#16#0000;
	_wAddDiagCode := WORD#16#0000;
	MEMSET(ADR(arrReadParameter),0,SIZEOF(arrReadParameter));
END_IF


// function blocks to read / write
_ReadParam(
			sNetId:= _sNetId, 
			nSlaveAddr:= _uintSlaveAddr, 
			nSubIndex:= 0, 
			nIndex:= _wIndex, 
			pDstBuf:= ADR(_arrReadBuffer), 
			cbBufLen:= _udintReadLength, 
			bExecute:= _xReadCommand, 
			tTimeout:= tTimeOutReading , 
			bBusy=> , 
			bError=> , 
			nErrId=> );	
			
_WriteParam(
			sNetId:= _sNetId, 
			nSlaveAddr:= _uintSlaveAddr, 
			nSubIndex:= 0 , 
			nIndex:= _wIndex, 
			pSrcBuf:= ADR(_arrWriteBuffer), 
			cbBufLen:= _udintSendLength, 
			bExecute:= _xWriteCommand, 
			tTimeout:= tTimeOutWriting , 
			bBusy=> , 
			bError=> , 
			nErrId=> );			


			

// Set Output data
	xActive := _xActive;
	xBusy := _xBusy;
	xError := _xError;
	wDiagCode := _wDiagCode;
	wAddDiagCode := _wAddDiagCode;

END_FUNCTION_BLOCK
